TYPE ST_INSTANCE_STATE :
STRUCT
  State     : E_INSTANCE_STATE;
  Progress  : E_PROGRESS;
END_STRUCT
END_TYPE

(* stored: Version 1.1.0.1, ProductVersion 3.1.4026.13
   DUT ST_INSTANCE_STATE: Id {25be858d-d916-4b39-b005-5bd8859b7f13} *)
